{attribute 'qualified_only'}
VAR_GLOBAL
	G_GlobalArry01 : ARRAY [0..99] OF INT;
	G_GlobalArry02 : ARRAY [0..99] OF INT;
	G_Cycle: INT:=1;
	G_Cycle2: int:=1;		
END_VAR

(* stored: Version 1.1.0.1, ProductVersion 3.1.4022.7
   GVL GlobalVar: Id {ea46ffc4-9a00-42e1-97c9-39dc96f90097} *)
